(* IEC 61131-3 sources: WarwickBoringPLC/Misc, 3 files *)

(* ---- ConsumptionMeterCalculator.FB.st ---- *)
// Calculates the rate for the consumption meter
FUNCTION_BLOCK ConsumptionMeterCalculator
VAR_INPUT
END_VAR
VAR_OUTPUT
END_VAR
VAR
	// Consumption meter triggers
	consumptionPulseTrigger : R_TRIG; (* to catch the rising signal edge *)
  	consumptionResetTrigger : R_TRIG; (* to catch the rising signal edge *)

	// Consumption meter rate calculation
	tDelta, tCurrent, tLast : TIME;

	impulseSize : REAL := 1000; // 1 pulse = 1 kWH, TO CHECK
END_VAR
consumptionPulseTrigger (CLK := mGVL.energyConsumptionPulse); (* finds the counting up events *)
consumptionResetTrigger (CLK := FALSE); (* finds the clear commands *) // TODO

IF consumptionPulseTrigger.Q
THEN
	// One impulse = 10L
	mainGVL.energyConsumptionTotal := mainGVL.energyConsumptionTotal + TO_INT(impulseSize);

	tCurrent := TO_TIME(SysTimeGetMs());

	// Calculate delta
	tDelta := tCurrent - tLast; // ms

	// Calculate rate
	mainGVL.energyConsumptionPower := impulseSize * 1000 / TIME_TO_REAL(tDelta) ; // w, x1000 as time is in ms.

	tLast := tCurrent;

END_IF;
IF consumptionResetTrigger.Q
	// Reset total energy consumption
	THEN mainGVL.energyConsumptionTotal := 0;
END_IF;

(* ---- TelemetryMQTT.FB.st ---- *)
// Sends the required telemetry to the supplied MQTT server
FUNCTION_BLOCK TelemetryMQTT
VAR_INPUT
END_VAR
VAR_OUTPUT
END_VAR
VAR
	MQTT_IN_OUT : MQTT.MQTT_IN_OUT;

	HandleMQTT : MQTT.MqttClient;

	PublishMQTT : MQTT.MQTTPublish;
	init : BOOL;
	doPublish : BOOL := FALSE;

	url : STRING := '192.168.0.133:1883';
	topic : STRING := 'topic';
	payloadString : STRING := 'Hello there';

END_VAR

HandleMQTT(

	MQTT_IN_OUT := MQTT_IN_OUT,
	ENABLE := TRUE,
	URL := url,
	TIMEOUT := T#1s,
	TLS := FALSE
);

IF NOT init THEN
	init := TRUE;
	PublishMQTT.SetMqttInOut(MQTT_IN_OUT := MQTT_IN_OUT);

END_IF

PublishMQTT(
	Topic := ADR(url),
	PayloadString := ADR(payloadString),
	PublishAsString := TRUE,
	QoSIn := MQTT.QoS.ExactlyOnce,
	MRetain := FALSE,
	send := visuGVL.meResetFlowMeter);

(* ---- PLC_MISC.st ---- *)
// Used to get misc PLC sensors and values
PROGRAM PLC_MISC
VAR
	result : POINTER TO CmpApp.RTS_IEC_RESULT;
END_VAR

mainGVL.cpuLoad := SchedGetProcessorLoad(result);
